(* Logix 5000 project; controller Safety vendor 1 type 14 code 148 rev 32.11; software revision 32.03; part 17 of 17 *)
(* tags used below, declared in another part *)
   A1_S20_ModFlt : ALIAS FOR Flt_Modules[0].0;   // A1 Point I/O Slot20 Module Fault (1 = Fault)
   A1_S21_ModFlt : ALIAS FOR Flt_Modules[0].1;   // A1 Point I/O Slot21 Module Fault (1 = Fault)
   C1_S12_ModFlt : ALIAS FOR Flt_Modules[0].2;   // C1 Point I/O Slot12 Module Fault (1 = Fault)
   CC : ALIAS FOR Diag_Tmp.0;   // Chris Como's Test Bit Always On Bit
   ChgMe : BOOL;
   CHPLC_S1_ModFlt : ALIAS FOR Flt_Modules[0].3;   // CHPLC Point I/O Slot01 Module Fault (1 = Fault)
   CHPLC_S2_ModFlt : ALIAS FOR Flt_Modules[0].4;   // CHPLC Point I/O Slot02 Module Fault (1 = Fault)
   CHPLC_S3_ModFlt : ALIAS FOR Flt_Modules[0].5;   // CHPLC Point I/O Slot03 Module Fault (1 = Fault)
   CHPLC_S4_ModFlt : ALIAS FOR Flt_Modules[0].6;   // CHPLC Point I/O Slot04 Module Fault (1 = Fault)
   CHPLC_S5_ModFlt : ALIAS FOR Flt_Modules[0].7;   // CHPLC Point I/O Slot05 Module Fault (1 = Fault)
   CHPLC_S6_ModFlt : ALIAS FOR Flt_Modules[0].8;   // CHPLC Point I/O Slot06 Module Fault (1 = Fault)
   Citect_HB_Flt : BOOL;   // Citect Heartbeat Fault ( 1= Fault)
   D1_S12_ModFlt : ALIAS FOR Flt_Modules[0].9;   // D1 Point I/O Slot12 Module Fault (1 = Fault)
   DAM : ALIAS FOR Diag_Tmp.4;   // Doug M Always Off Test Bit
   Darin_M_Safety_Test_Bit : BOOL;
   Diag_Tmp : DINT;   // Temp Bit Test Bit
   DPD_S14_ModFlt : ALIAS FOR Flt_Modules[0].10;   // DPD Point I/O Slot14 Module Fault (1 = Fault)
   DPD_S15_ModFlt : ALIAS FOR Flt_Modules[0].11;   // DPD Point I/O Slot15 Module Fault (1 = Fault)
   E1_S10_ModFlt : ALIAS FOR Flt_Modules[0].12;   // E1 Point I/O Slot10 Module Fault (1 = Fault)
   F1_S19_ModFlt : ALIAS FOR Flt_Modules[0].13;   // F1 Point I/O Slot19 Module Fault (1 = Fault)
   F1_S20_ModFlt : ALIAS FOR Flt_Modules[0].14;   // F1 Point I/O Slot20 Module Fault (1 = Fault)
   FUTURE : ALIAS FOR Diag_Tmp.1;   // FUTURE
   G1_S11_ModFlt : ALIAS FOR Flt_Modules[0].15;   // G1 Point I/O Slot11 Module Fault (1 = Fault)
   G1_S12_ModFlt : ALIAS FOR Flt_Modules[0].16;   // G1 Point I/O Slot12 Module Fault (1 = Fault)
   H1_S5_ModFlt : ALIAS FOR Flt_Modules[0].17;   // H1 Point I/O Slot05 Module Fault (1 = Fault)
   H1_S6_ModFlt : ALIAS FOR Flt_Modules[0].18;   // H1 Point I/O Slot06 Module Fault (1 = Fault)
   Machine_HB_Flt : BOOL;   // Machine Heartbeat Fault ( 1= Fault)
   MCC1_S1_ModFlt : ALIAS FOR Flt_Modules[2].0;   // MCC1 Point I/O Slot01 Module Fault (1 = Fault)
   MCC1_S6_ModFlt : ALIAS FOR Flt_Modules[2].1;   // MCC1 Point I/O Slot06 Module Fault (1 = Fault)
   MCC2_S1_ModFlt : ALIAS FOR Flt_Modules[2].2;   // MCC2 Point I/O Slot01 Module Fault (1 = Fault)
   MCC2_S2_ModFlt : ALIAS FOR Flt_Modules[2].3;   // MCC2 Point I/O Slot02 Module Fault (1 = Fault)
   MCC3_S1_ModFlt : ALIAS FOR Flt_Modules[2].4;   // MCC3 Point I/O Slot01 Module Fault (1 = Fault)
   MCC3_S3_ModFlt : ALIAS FOR Flt_Modules[2].5;   // MCC3 Point I/O Slot03 Module Fault (1 = Fault)
   MCC3_S4_ModFlt : ALIAS FOR Flt_Modules[2].6;   // MCC3 Point I/O Slot04 Module Fault (1 = Fault)
   MCC4_S1_ModFlt : ALIAS FOR Flt_Modules[2].7;   // MCC4 Point I/O Slot01 Module Fault (1 = Fault)
   MCC4_S3_ModFlt : ALIAS FOR Flt_Modules[2].8;   // MCC4 Point I/O Slot03 Module Fault (1 = Fault)
   MCC4_S4_ModFlt : ALIAS FOR Flt_Modules[2].9;   // MCC4 Point I/O Slot04 Module Fault (1 = Fault)
   MCC5_S1_ModFlt : ALIAS FOR Flt_Modules[2].10;   // MCC5 Point I/O Slot01 Module Fault (1 = Fault)
   MCC5_S3_ModFlt : ALIAS FOR Flt_Modules[2].11;   // MCC5 Point I/O Slot03 Module Fault (1 = Fault)
   MCC5_S4_ModFlt : ALIAS FOR Flt_Modules[2].12;   // MCC5 Point I/O Slot04 Module Fault (1 = Fault)
   MCC5_S5_ModFlt : ALIAS FOR Flt_Modules[2].13;   // MCC5 Point I/O Slot05 Module Fault (1 = Fault)
   OS11_S1_ModFlt : ALIAS FOR Flt_Modules[1].11;   // OS11 Point I/O Slot01 Module Fault (1 = Fault)
   OS13_S1_ModFlt : ALIAS FOR Flt_Modules[1].12;   // OS13 Point I/O Slot01 Module Fault (1 = Fault)
   OS14_S1_ModFlt : ALIAS FOR Flt_Modules[1].13;   // OS14 Point I/O Slot01 Module Fault (1 = Fault)
   OS15_S1_ModFlt : ALIAS FOR Flt_Modules[1].14;   // OS15 Point I/O Slot01 Module Fault (1 = Fault)
   OS16_S1_ModFlt : ALIAS FOR Flt_Modules[1].15;   // OS16 Point I/O Slot01 Module Fault (1 = Fault)
   OS1_S1_ModFlt : ALIAS FOR Flt_Modules[1].0;   // OS1 Point I/O Slot01 Module Fault (1 = Fault)
   OS2_S1_ModFlt : ALIAS FOR Flt_Modules[1].1;   // OS2 Point I/O Slot01 Module Fault (1 = Fault)
   OS3_S1_ModFlt : ALIAS FOR Flt_Modules[1].2;   // OS3 Point I/O Slot01 Module Fault (1 = Fault)
   OS4N_S1_ModFlt : ALIAS FOR Flt_Modules[1].3;   // OS4N Point I/O Slot01 Module Fault (1 = Fault)
   OS4S_S1_ModFlt : ALIAS FOR Flt_Modules[1].5;   // OS4S Point I/O Slot01 Module Fault (1 = Fault)
   OS5_S1_ModFlt : ALIAS FOR Flt_Modules[1].7;   // OS5 Point I/O Slot01 Module Fault (1 = Fault)
   OS6_S1_ModFlt : ALIAS FOR Flt_Modules[1].8;   // OS6 Point I/O Slot01 Module Fault (1 = Fault)
   OS8_S1_ModFlt : ALIAS FOR Flt_Modules[1].9;   // OS8 Point I/O Slot01 Module Fault (1 = Fault)
   OS9_S1_ModFlt : ALIAS FOR Flt_Modules[1].10;   // OS9 Point I/O Slot01 Module Fault (1 = Fault)
   SDPLC_S1_ModFlt : ALIAS FOR Flt_Modules[0].19;   // SDPLC Point I/O Slot01 Module Fault (1 = Fault)
   SDPLC_S2_ModFlt : ALIAS FOR Flt_Modules[0].20;   // SDPLC Point I/O Slot02 Module Fault (1 = Fault)
   Sfty_InstrFlts0_CTC : BOOL;   // Coil To Coil Estop Safety Instructions OK ( 1= No Faults)
   Sfty_InstrFlts0_CTL : BOOL;   // Cut To Length Estop Safety Instructions OK ( 1= No Faults)
   Sfty_InstrFlts0_Total : BOOL;   // Total Mode Estop Safety Instructions OK ( 1= No Faults)
   Sfty_InstrFlts1_CTC : BOOL;   // Coil To Coil Safe-Off Safety Instructions OK ( 1= No Faults)
   Sfty_InstrFlts1_CTL : BOOL;   // Cut To Length Safe-Off Safety Instructions OK ( 1= No Faults)
   Sfty_InstrFlts1_Total : BOOL;   // Total Mode Safe-Off Safety Instructions OK ( 1= No Faults)
   Sfty_InstrFlts2_CTC : BOOL;   // Coil To Coil FVR/FVNR Starters Safety Instructions OK ( 1= No Faults)
   Sfty_InstrFlts2_CTL : BOOL;   // Cut To Length FVR/FVNR Starters Safety Instructions OK ( 1= No Faults)
   Sfty_InstrFlts2_Total : BOOL;   // Total Mode FVR/FVNR Starters Safety Instructions OK ( 1= No Faults)
   Sfty_ModFlts0_CTC : BOOL;   // Coil To Coil General I/O Safety Module Faults ( 1= OK)
   Sfty_ModFlts0_CTL : BOOL;   // Cut To Length General I/O Safety Module Faults ( 1= OK)
   Sfty_ModFlts0_Total : BOOL;   // Total Mode General I/O Safety Module Faults ( 1= OK)
   Sfty_ModFlts1_CTC : BOOL;   // Coil To Coil Operator Station Safety Module Faults ( 1= OK)
   Sfty_ModFlts1_CTL : BOOL;   // Cut To Length Operator Station Safety Module Faults ( 1= OK)
   Sfty_ModFlts1_Total : BOOL;   // Total Mode Operator Station Safety Module Faults ( 1= OK)
   Sfty_ModFlts2_CTC : BOOL;   // Coil To Coil MCC Safety Module Faults ( 1= OK)
   Sfty_ModFlts2_CTL : BOOL;   // Cut To Lenght MCC Safety Module Faults ( 1= OK)
   Sfty_ModFlts2_Total : BOOL;   // Total Mode MCC Safety Module Faults ( 1= OK)
   Shear_HB_Flt : BOOL;   // Shear Heartbeat Fault ( 1= Fault)
   VS2_S10_ModFlt : ALIAS FOR Flt_Modules[0].21;   // VS2 Point I/O Slot10 Module Fault (1 = Fault)
(* System, continued *)

ROUTINE MainRoutine   (* ladder *)
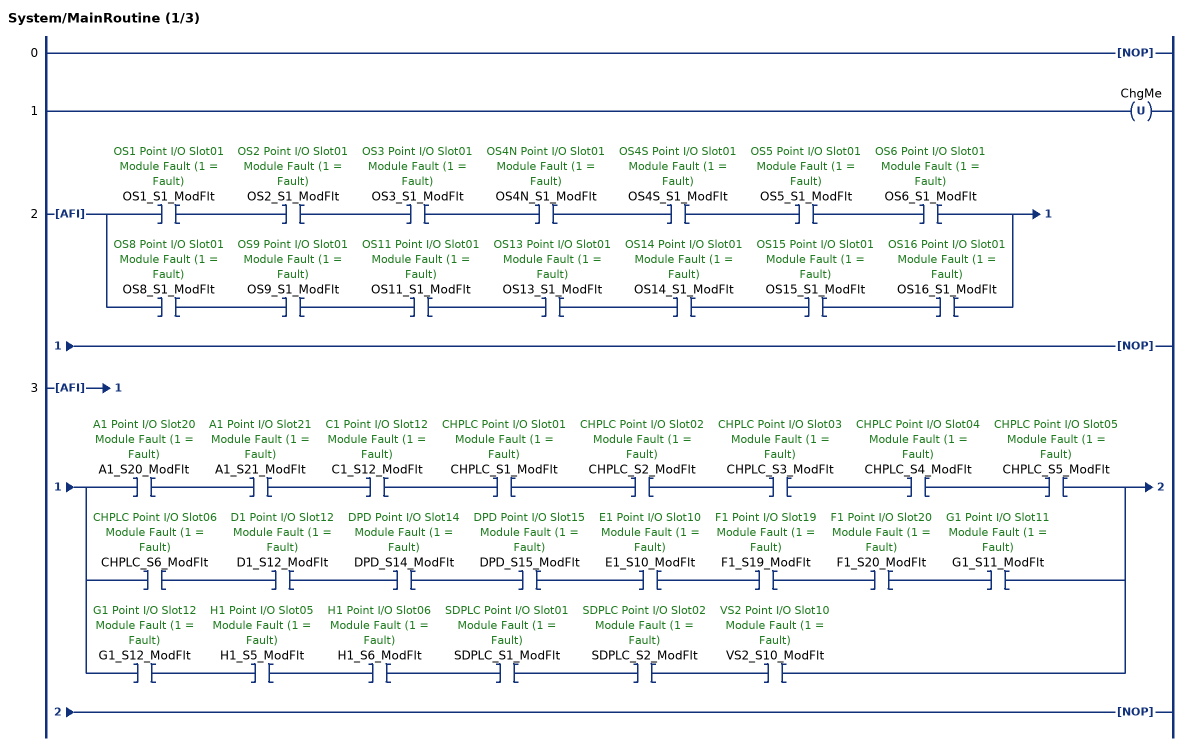
   0: NOP();
   1: OTU(ChgMe);
   2: AFI()[XIC(OS1_S1_ModFlt) XIC(OS2_S1_ModFlt) XIC(OS3_S1_ModFlt) XIC(OS4N_S1_ModFlt) XIC(OS4S_S1_ModFlt) XIC(OS5_S1_ModFlt) XIC(OS6_S1_ModFlt) ,XIC(OS8_S1_ModFlt) XIC(OS9_S1_ModFlt) XIC(OS11_S1_ModFlt) XIC(OS13_S1_ModFlt) XIC(OS14_S1_ModFlt) XIC(OS15_S1_ModFlt) XIC(OS16_S1_ModFlt) ]NOP();
   3: AFI()[XIC(A1_S20_ModFlt) XIC(A1_S21_ModFlt) XIC(C1_S12_ModFlt) XIC(CHPLC_S1_ModFlt) XIC(CHPLC_S2_ModFlt) XIC(CHPLC_S3_ModFlt) XIC(CHPLC_S4_ModFlt) XIC(CHPLC_S5_ModFlt) ,XIC(CHPLC_S6_ModFlt) XIC(D1_S12_ModFlt) XIC(DPD_S14_ModFlt) XIC(DPD_S15_ModFlt) XIC(E1_S10_ModFlt) XIC(F1_S19_ModFlt) XIC(F1_S20_ModFlt) XIC(G1_S11_ModFlt) ,XIC(G1_S12_ModFlt) XIC(H1_S5_ModFlt) XIC(H1_S6_ModFlt) XIC(SDPLC_S1_ModFlt) XIC(SDPLC_S2_ModFlt) XIC(VS2_S10_ModFlt) ]NOP();
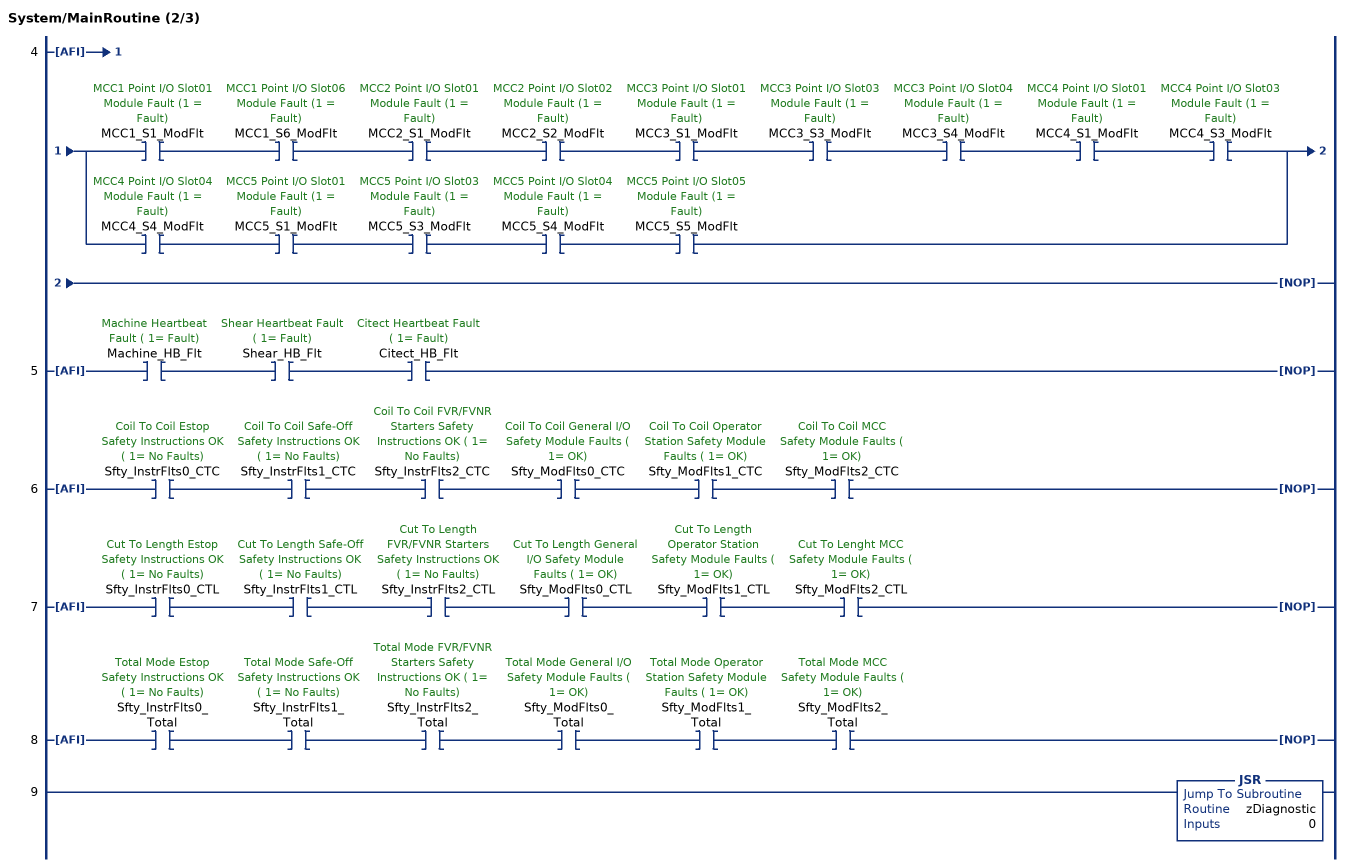
   4: AFI()[XIC(MCC1_S1_ModFlt) XIC(MCC1_S6_ModFlt) XIC(MCC2_S1_ModFlt) XIC(MCC2_S2_ModFlt) XIC(MCC3_S1_ModFlt) XIC(MCC3_S3_ModFlt) XIC(MCC3_S4_ModFlt) XIC(MCC4_S1_ModFlt) XIC(MCC4_S3_ModFlt) ,XIC(MCC4_S4_ModFlt) XIC(MCC5_S1_ModFlt) XIC(MCC5_S3_ModFlt) XIC(MCC5_S4_ModFlt) XIC(MCC5_S5_ModFlt) ]NOP();
   5: AFI()XIC(Machine_HB_Flt)XIC(Shear_HB_Flt)XIC(Citect_HB_Flt)NOP();
   6: AFI()XIC(Sfty_InstrFlts0_CTC)XIC(Sfty_InstrFlts1_CTC)XIC(Sfty_InstrFlts2_CTC)XIC(Sfty_ModFlts0_CTC)XIC(Sfty_ModFlts1_CTC)XIC(Sfty_ModFlts2_CTC)NOP();
   7: AFI()XIC(Sfty_InstrFlts0_CTL)XIC(Sfty_InstrFlts1_CTL)XIC(Sfty_InstrFlts2_CTL)XIC(Sfty_ModFlts0_CTL)XIC(Sfty_ModFlts1_CTL)XIC(Sfty_ModFlts2_CTL)NOP();
   8: AFI()XIC(Sfty_InstrFlts0_Total)XIC(Sfty_InstrFlts1_Total)XIC(Sfty_InstrFlts2_Total)XIC(Sfty_ModFlts0_Total)XIC(Sfty_ModFlts1_Total)XIC(Sfty_ModFlts2_Total)NOP();
   9: JSR(zDiagnostic,0);
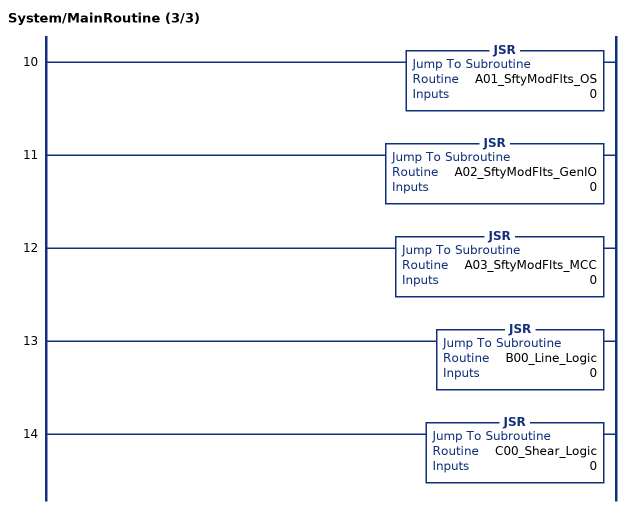
   10: JSR(A01_SftyModFlts_OS,0);
   11: JSR(A02_SftyModFlts_GenIO,0);
   12: JSR(A03_SftyModFlts_MCC,0);
   13: JSR(B00_Line_Logic,0);
   14: JSR(C00_Shear_Logic,0);
END_ROUTINE

ROUTINE zDiagnostic   (* ladder *)
// Diagnostics
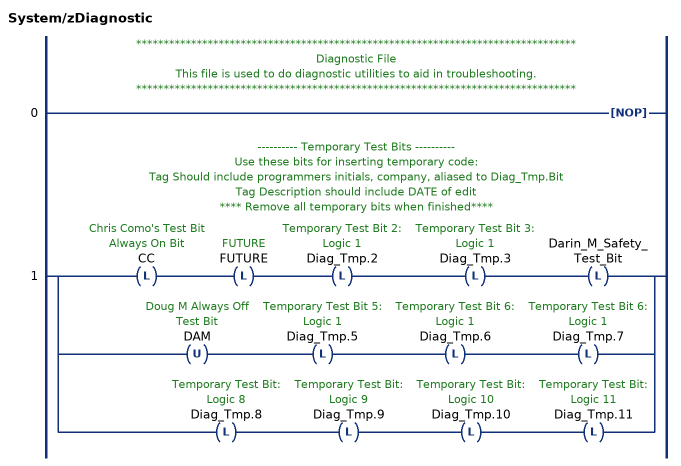
   // ********************************************************************************
   // 			Diagnostic File
   // This file is used to do diagnostic utilities to aid in troubleshooting.
   // ********************************************************************************
   0: NOP();
   // ---------- Temporary Test Bits ----------
   // Use these bits for inserting temporary code:
   // Tag Should include programmers initials, company, aliased to Diag_Tmp.Bit
   // Tag Description should include DATE of edit
   // **** Remove all temporary bits when finished****
   1: [OTL(CC) OTL(FUTURE) OTL(Diag_Tmp.2) OTL(Diag_Tmp.3) OTL(Darin_M_Safety_Test_Bit) ,OTU(DAM) OTL(Diag_Tmp.5) OTL(Diag_Tmp.6) OTL(Diag_Tmp.7) ,OTL(Diag_Tmp.8) OTL(Diag_Tmp.9) OTL(Diag_Tmp.10) OTL(Diag_Tmp.11) ];
END_ROUTINE
END_PROGRAM
